FUNCTION_BLOCK FB_FileLogger IMPLEMENTS  I_Logger
VAR
END_VAR

{warning 'add method implementation '}
METHOD M_Log : BOOL
VAR_INPUT
	sMessage	: STRING(255);
END_VAR
ADSLOGSTR(
			msgCtrlMask:= ADSLOG_MSGTYPE_ERROR,
			msgFmtStr := 'File Log: %s',
			strArg := sMessage );
END_METHOD

END_FUNCTION_BLOCK

(* stored: Version 1.1.0.1, ProductVersion 3.1.4024.16
   POU FB_FileLogger: Id {70e13956-18a1-4a1a-8300-b10668faf7f2}, SpecialFunc None
   Method M_Log: Id {502db601-b68a-481a-a48d-fe6f6f65a7ae} *)
